PROGRAM P_red
VAR
	a,b,c:INT;
END_VAR

c:=a*b;

END_PROGRAM

(* stored: Version 1.1.0.1, ProductVersion 3.1.4024.11
   POU P_red: Id {5e5ffa00-0b90-446e-8e31-cef0c919759a}, SpecialFunc None *)
